(* PLC project Wiring, CODESYS V3.5 SP8 Patch 2 *)
(* stored: creationDateTime 1990-01-12T12:00:00, modificationDateTime 1990-01-12T12:12:12 *)

PROGRAM WIRING

          	
%MX3.3 := %IX0.0;
 
%MX0.0 := %IX0.1;
 
			
          
END_PROGRAM
